ABB RobotStudio station: Airhockey2.0.rspag

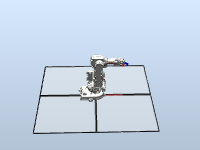
--- station ---
Station Airhockey2.0 (saved by RobotStudio format 3)
Controller IRB_140_6kg_0.81m
  mechanical unit ROB_1: IRB140_6_81_C_03, 6 joints, base frame (0, 0, 0) mm
Layout (positions relative to the parent item):
  - IRB140_6_81_C_03 [mechanism, from Robots\IRB140_6_81_C_G_03.rslib] at (0, 0, 0) mm; joint values [0, 0, 0, 0, 0.5236, 0] (rad or m)

--- Backups/IRB_140_6kg_0.81m/RAPID/TASK1/PROGMOD/CalibData.mod ---
MODULE CalibData
    CONST num xMin:=0;
    CONST num xMax:= 260;
    CONST num xMaxMitte:=386;
    CONST num yMin:= 0;
    CONST num yMax:= 690;
	TASK PERS wobjdata Workobject_Table:=[FALSE,TRUE,"",[[0,0,0],[1,0,0,0]],[[423.6,-349.4,294.7],[1,0,0,0]]];
    CONST robtarget Target_10:=[[xMin,yMin,30],[0,1,0,0],[-1,0,0,0],[9E9,9E9,9E9,9E9,9E9,9E9]];
    CONST robtarget Target_20:=[[xMin,yMax,30],[0,1,0,0],[-1,0,0,0],[9E9,9E9,9E9,9E9,9E9,9E9]];
    CONST robtarget Target_30:=[[xMax,yMax,30],[0,1,0,0],[-1,0,0,0],[9E9,9E9,9E9,9E9,9E9,9E9]];
    CONST robtarget Target_40:=[[xMax,yMin,30],[0,1,0,0],[-1,0,0,0],[9E9,9E9,9E9,9E9,9E9,9E9]];
    CONST robtarget Target_Home:=[[453,26,610],[0,1,0,0],[-1,0,0,0],[9E9,9E9,9E9,9E9,9E9,9E9]];
ENDMODULE

--- Backups/IRB_140_6kg_0.81m/RAPID/TASK1/PROGMOD/positionenAbfahren.mod ---
MODULE positionenAbfahren

VAR socketdev server_socket;
VAR socketdev client_socket;
VAR socketdev my_socket;
VAR string receive_string;
VAR string client_ip;
VAR string partX;
VAR string partY;
VAR robtarget Target;
VAR num count;
VAR num x := 0;
VAR num y := 345;
VAR num z := 0;
VAR num found;
VAR num xMaxV;
VAR bool okX;
VAR bool okY;




PROC main()

Target:=[[x,y,z],[0,1,0,0],[-1,0,0,0],[9E9,9E9,9E9,9E9,9E9,9E9]];
MoveL Target,v5000,fine,tool0\WObj:=Workobject_Table;

SocketCreate my_socket;
SocketConnect my_socket,"192.168.28.222", 1025 \Time:=WAIT_MAX;


WHILE (TRUE) DO

!Empfange Daten
SocketReceive my_socket \Str:= receive_string \Time:=WAIT_MAX;


found := StrFind(receive_string,1,";");

IF (found>StrLen(receive_string)) THEN
    ErrWrite \W, "Trennzeichen nicht gefunden","Koordinten müssen durch ; getrennt werden";
    GOTO abbrechen;
ENDIF

!Auslesen der Koordinten als String
partX := StrPart(receive_string,1,found-1);
partY := StrPart(receive_string,found+1,StrLen(receive_string)-found);

!Convertieren in Zahlen
okX := StrToVal(partX,x);
okY := StrToVal(partY,y);

!Ueberpruefung, ob Convertierung funktioniert hat
IF NOT (okX AND okY) THEN
    ErrWrite \W, "Zeichenfolge konnte nicht in eine Zahl umgewandelt werden", "";
    GOTO abbrechen;
ENDIF

!TPWrite " " \Num:=x;
!TPWrite " " \Num:=y;

!Ueberpruefung, ob Koordinaten außerhalb des Spielfeldes liegen
IF abs(y-345)<1 THEN
    xMaxV:= xMaxMitte;
ELSE
    xMaxV:= xMax;
ENDIF

IF (x<xMin) OR (x>xMaxV) OR (y<yMin) OR (y>yMax) THEN
    ErrWrite \W, "Gesendete Koordinaten liegen außerhalb des Spielfeldes" , receive_string;
    GOTO abbrechen;
ENDIF

!Bewegungsanweisung an Roboter
Target:=[[x,y,z],[0,1,0,0],[-1,0,0,0],[9E9,9E9,9E9,9E9,9E9,9E9]];
MoveL Target,vMax,fine,tool0\WObj:=Workobject_Table;


abbrechen:
SocketSend my_socket \Str:="Ready";

ENDWHILE


ERROR
RETRY;
UNDO
SocketClose my_socket;

	ENDPROC

	PROC Jump_Home()
        MoveL Target_Home,v50,fine,tool0\WObj:=wobj0;
    ENDPROC

    PROC Kalibrierungstest()
	    MoveL Target_10,v50,fine,tool0\WObj:=Workobject_Table;
        MoveL Target_20,v50,fine,tool0\WObj:=Workobject_Table;
        MoveL Target_30,v50,fine,tool0\WObj:=Workobject_Table;
        MoveL Target_40,v50,fine,tool0\WObj:=Workobject_Table;

	ENDPROC



ENDMODULE

--- Backups/IRB_140_6kg_0.81m/RAPID/TASK1/SYSMOD/LINKEDM.sys ---
%%%
  VERSION:1
  LANGUAGE:ENGLISH
%%%

MODULE LINKEDM (SYSMODULE)

! FOLLOWER
!     Name of electronically linked follower axis used by operator at teach pendent.
      PERS string l_f_axis_name{5}       :=  ["",  "", "", "", ""];

!     Name of the mechanical unit for follower axis.
      PERS string l_f_mecunt_n{5}  :=  ["", "", "", "", ""];

!     Linked follower axis number in the mechanical unit (first axis in mech. unit is number 1).
      PERS num l_f_axis_no{5}      :=  [0,          0,   0,  0,  0];

! MASTER
!     Name of the mechanical unit for linked master axis.
      PERS string l_m_mecunt_n{5} :=  ["", "", "", "", ""];

!     Linked master axis number in the mechanical unit (first axis in mech. unit is number 1).
!     See axis number table in documentation for different master mechanical units.
      PERS num l_m_axis_no{5}     :=  [0,  0,  0,  0,  0];

! POSITION OFFSET
!     The increase of the allowed offset position between the master and follower
!     positions, used when starting AUTO mode. As soon as the offset is decreased
!     the old configurated parameter is used.
!     Example: 3 => the configurated value of allowed offset is increased 3 times.
      PERS num offset_ratio{5}       :=  [10,  10,   10,  10,  10];

! SPEED RATIO
!     Speed_ratio used in AUTO and JOG modes [ very_slow   slow    normal    fast]
!     Value 1 = max allowed manual speed.
      CONST num speed_ratio {20}      := [0.01, 0.01, 0.01, 0.01, 0.01,
                                          0.05, 0.05, 0.05, 0.05, 0.05,
                                          0.20, 0.20, 0.20, 0.20, 0.20,
                                          1.00, 1.00, 1.00, 1.00, 1.00];

! STEP SIZE
!     Displacement position used in JOG mode for each activation of positive or
!     negative movement.                  [very_short    short   normal   long]
!     Unit degees or meter.
      CONST num displacement {20}     := [0.001, 0.001, 0.001, 0.001, 0.001,
                                          0.005, 0.005, 0.005, 0.005, 0.005,
                                          0.020, 0.020, 0.020, 0.020, 0.020,
                                          0.100, 0.100, 0.100, 0.100, 0.100];


!-------------------------------------------------------------
 PROC Linked_m ()
      Linked_m_exe ;
 ENDPROC
ENDMODULE
